ADAPTER L3_ASetup
  (* Standard: 61499-1 *)
  (* Version 0.0, 2008-04-22, EQUEROL, UJI *)
  (* Version 1.0, 2015-01-08, EQUEROL, UJI, modified output data *)
  (* Version 2.0, 2015-03-13, EQUEROL, UJI *)
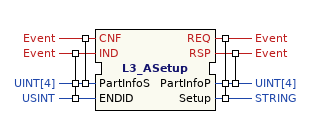
  EVENT_INPUT
    CNF WITH PartInfoS; (* Setup assignation confirmation *)
    IND WITH PartInfoS, ENDID; (* Completed setup indication *)
  END_EVENT
  EVENT_OUTPUT
    REQ WITH PartInfoP, Setup; (* Plugin request to assign a setup *)
    RSP WITH PartInfoP; (* Completed setup indication treatement resposne *)
  END_EVENT
  VAR_INPUT
    PartInfoS : ARRAY [0..3] OF UINT; (* Part ID, Part Family, Part Type, MID *)
    ENDID : USINT; (* Setup execution returned code *)
  END_VAR
  VAR_OUTPUT
    PartInfoP : ARRAY [0..3] OF UINT; (* PartID, Part Family, Part Type, MID *)
    Setup : STRING; (* Subphase to be transmitted *)
  END_VAR
  SERVICE SOCKET/PLUG
    SEQUENCE request_confirm
      SOCKET.REQ(REQD) -> PLUG.REQ(REQD);
      PLUG.CNF(CNFD) -> SOCKET.CNF(CNFD);
    END_SEQUENCE
    SEQUENCE indication_response
      PLUG.IND(INDD) -> SOCKET.IND(INDD);
      SOCKET.RSP(RSPD) -> PLUG.RSP(RSPD);
    END_SEQUENCE
  END_SERVICE
END_ADAPTER
